Yaskawa INFORM job: TRIAL.JBI

/JOB
//NAME TRIAL
//POS
///NPOS 12,0,0,0,0,0
///TOOL 0
///POSTYPE PULSE
///PULSE
C00000=-77498,-145772,-106573,97596,-115753,-139143
C00001=-77498,-145772,-106573,97596,-115753,-139143
C00002=-132135,-154754,-108505,82259,-80313,-137071
C00003=-129638,-121031,-104437,85498,-80265,-145701
C00004=-127515,-118285,-96743,74295,-83753,-143626
C00005=-122949,-124554,-111252,75325,-85737,-146264
C00006=-154535,-123515,-134589,197689,-98247,-50314
C00007=-154533,-111372,-118101,197836,-88793,-50634
C00008=-151578,-99997,-113617,197702,-91633,-48954
C00009=-150626,-99695,-112249,197648,-90930,-55708
C00010=-148795,-77316,-101056,197639,-96208,-63152
C00011=-135154,-87084,-109017,196538,-92557,-58265
//INST
///DATE 2022/04/06 09:35
///ATTR SC,RW
///GROUP1 RB1
NOP
MOVJ C00000 VJ=65.00
MOVL C00001 V=150.0
MOVL C00002 V=150.0
MOVL C00003 V=150.0
MOVL C00004 V=150.0
MOVL C00005 V=150.0  //AWAY
MOVL C00006 V=150.0
MOVL C00007 V=150.0
MOVL C00008 V=150.0
MOVL C00009 V=150.0
MOVL C00010 V=150.0
MOVL C00011 V=150.0  //AWAY
END
